Staubli VAL3: JointStateMsg.dtx

public Header header
  [0]
    num nMsgType
    num nCommType
    num nReplyCode
    num nData[12]
public Body body
  [0]
    num nData[44]
public JointState jointState
  [0]
    num nSeq
    num nJoints[10]
public Prefix prefix
  [0]
    num nLength
    num nData[4]
